INTERFACE I_Graph EXTENDS I_BaseElement, I_HaveNodes

METHOD PUBLIC Accept
VAR_INPUT
	Visitor : I_GraphVisitor;
END_VAR
END_METHOD

METHOD PUBLIC Clear
VAR_INPUT
END_VAR
END_METHOD

METHOD PUBLIC GetCurrentUuid : Uuid
VAR_INPUT
END_VAR
END_METHOD

METHOD PUBLIC GetNodes : I_Nodes
VAR_INPUT
END_VAR
END_METHOD

METHOD Run
VAR_INPUT
END_VAR
END_METHOD

END_INTERFACE

(* stored: Version 1.1.0.1, ProductVersion 3.1.4024.12
   Itf I_Graph: Id {45c251a4-de8e-0c6c-2a3e-8a87e382a116}
   Method Accept: Id {255392e5-cd9d-0e73-21a1-ba770a89b900}
   Method Clear: Id {7d56e05b-0642-0e1a-2d09-f7343732854e}
   Method GetCurrentUuid: Id {95f60cde-6a93-08ea-19d9-a52bd39c68e0}
   Method GetNodes: Id {e673abbf-5566-0889-0a5c-d05bfe265452}
   Method Run: Id {60905f56-31e2-0c62-2fd4-d291a9b07dea} *)
